Fanuc KAREL source: ka00225.KL

-- PROVISIONAL review KL for V940-1; original PC SHA256 753682f55501feeac4ab5c1de32d6e4cbdc8ec420a2bfb57b8a0ae93f694d722
-- Incomplete behavior may be omitted. Consult companion uncertainty JSON. Do not deploy.
PROGRAM KA00225
%NOLOCKGROUP
BEGIN
  -- V9_COMPOSED_GLOBAL_TRANSFER_HINT repetitions=1; address IDs observed; pairing/direction/source/runtime held
  -- V9_TWO_GLOBAL_ADDRESS_COPY_HINT bounded five-record physical form; type/direction/source/runtime held
  -- V9_ZERO_TABLE_METADATA_HINT layout=0001; no indexed target words; source/name/runtime held
  -- UNRESOLVED_PC offsets 5-19; opcodes 22,22,1E
  -- UNRESOLVED_PC offsets 24-28; opcodes 7F
END KA00225
